FUNCTION_BLOCK FB_SELECT (* ANY Selection (Inputs & Outputs must be consistent) *)
  (* Standard: 61499-1-D.1; Classification: Selection Functions *)
  (* Version 0.0, 2002-04-10, JHC, Rockwell Automation *)
  (* Compiler header: package fb.rt.math; *)
  (* Compiler Java IBM VisualAge 3.0 *)
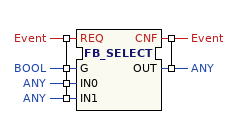
  EVENT_INPUT
    REQ WITH G, IN0, IN1;
  END_EVENT
  EVENT_OUTPUT
    CNF WITH OUT;
  END_EVENT
  VAR_INPUT
    G : BOOL; (* Selector *)
    IN0 : ANY; (* Selected when G=0 *)
    IN1 : ANY; (* Selected when G=1 *)
  END_VAR
  VAR_OUTPUT
    OUT : ANY; (* Selected value *)
  END_VAR
END_FUNCTION_BLOCK
